{attribute 'GeneratedUsingTerminal: EL6201-0000-0017'}
{attribute addProperty BoxType "EL6201-0000-0017"}
{attribute addProperty Id "Slave_5A_DI0BOOL1Slave_5A_DI1BOOL1Slave_5A_DI2BOOL1Slave_5A_DI3BOOL1Slave_5B_DI0BOOL1Slave_5B_DI1BOOL1Slave_5B_DI2BOOL1Slave_5B_DI3BOOL1"}
{attribute addProperty CRC "1134263989"}
{attribute addProperty Size "8"}
TYPE Slave_5_Inputs_439B7EB5 :
STRUCT
	{attribute addProperty Name "Slave_5A_DI0"}
	Slave_5A_DI0 : BOOL;
	{attribute addProperty Name "Slave_5A_DI1"}
	Slave_5A_DI1 : BOOL;
	{attribute addProperty Name "Slave_5A_DI2"}
	Slave_5A_DI2 : BOOL;
	{attribute addProperty Name "Slave_5A_DI3"}
	Slave_5A_DI3 : BOOL;
	{attribute addProperty Name "Slave_5B_DI0"}
	Slave_5B_DI0 : BOOL;
	{attribute addProperty Name "Slave_5B_DI1"}
	Slave_5B_DI1 : BOOL;
	{attribute addProperty Name "Slave_5B_DI2"}
	Slave_5B_DI2 : BOOL;
	{attribute addProperty Name "Slave_5B_DI3"}
	Slave_5B_DI3 : BOOL;
END_STRUCT
END_TYPE

(* stored: Version 1.2.0.0, ProductVersion 3.1.4024.9
   DUT Slave_5_Inputs_439B7EB5: Id {aed1062c-982c-42f3-834f-94130ee51111} *)
